PROGRAM MAIN
VAR
END_VAR

END_PROGRAM

(* stored: Version 1.1.0.1
   POU MAIN: Id {88a55e1a-3981-42a5-9f30-8c2daf9756cc} *)
